TYPE "UDT_ZC_DISP_FF"
VERSION : 0.1
   STRUCT
      Estado_SalidaFlip : Bool;   // Salida FLIP
      Estado_SalidaFlop : Bool;   // Salida FLOP
      Orden_Reset : Bool;   // Resetear estado de acumuladores
      Orden_Activar : Bool;   // Orden Marcha
      Orden_Pausa : Bool;   // Orden pausa
      Aux_FlipActivo : Bool;
      Aux_FlopActivo : Bool;
      Aux_Flanco : Bool;
      Config_SetPointTiempoFlip : Int;   // Tiempo Flip
      Config_SetPointTiempoFlop : Int;   // Tiempo Flop
      Aux_TiempoFlip : Int;   // Tiempo acumulador Flip
      Aux_TiempoFlop : Int;   // Tiempo acumulador Flop
   END_STRUCT;

END_TYPE

